// TIA Portal V18 export
// export: Created 2026-06-08T16:32:20.6513402Z, ExportSetting WithDefaults, DisplayName Totally Integrated Automation Portal, DisplayVersion V18, DisplayName TIA Portal Openness, DisplayVersion V18, DisplayName TIA Portal Version Control Interface, DisplayVersion V18, DisplayName STEP 7 Professional, DisplayVersion V18, DisplayName STEP 7 Safety, DisplayVersion V18, DisplayName WinCC Professional, DisplayVersion V18
DATA_BLOCK "LID PRODUCTION_DB"   // DB13
VERSION : 0.1
// stored: AutoNumber true, InstanceOfName LID PRODUCTION, InstanceOfType FB
"LID PRODUCTION"
BEGIN
END_DATA_BLOCK
